PROGRAM SavePersistentVariables 
VAR
	WritePersistentDataFB : WritePersistentData;  //WritePersistentData FunctionBlock
	StartTON : TON;
	IntervalTON :TON;
END_VAR
VAR // added by the converter: edge detectors and wires of the graphical bodies
    _rt1 : R_TRIG;
END_VAR

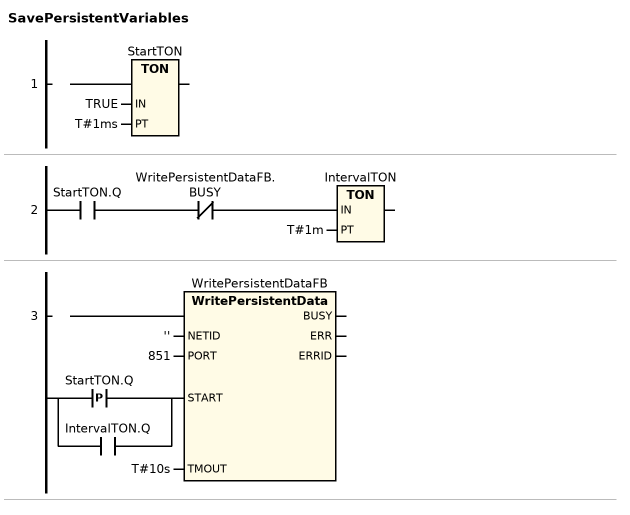
// NETWORK 1
StartTON(IN := TRUE, PT := T#1ms); // TON

// NETWORK 2
IntervalTON(IN := StartTON.Q AND NOT WritePersistentDataFB.BUSY, PT := T#1m); // TON

// NETWORK 3
_rt1(CLK := StartTON.Q);
WritePersistentDataFB(NETID := '', PORT := 851, START := _rt1.Q OR IntervalTON.Q, TMOUT := T#10s); // WritePersistentData

END_PROGRAM

(* stored: Version 1.1.0.1, ProductVersion 3.1.4020.12
   POU SavePersistentVariables: Id {c67a3f74-832b-476c-a1e6-509ff3032593}, SpecialFunc None *)
